Staubli VAL3: LEFTPOS.pgx

public program leftPos(string x_sItem, num x_nLength, string& x_sResult[])
  local num i
  local num l_nLength
  local string l_sItem
begin
  //-----------------------------------------------------------------------
  //Header begin
  //Description of program
  //  This program allows to keep x_nLength characters of a string from
  //  the left side.
  //  The characters after x_nLength on the right side will be truncated.
  //
  //Input parameters
  //  string x_sItem :
  //    role : string that you wan to cut
  //  num x_nLength :
  //    role : Length of the characters that you want to keep
  //
  //Output parameters
  //  string x_sResult :
  //    role : string truncated
  //
  //Example
  //  call leftPos("Staubli Robotics",7,sResult)
  //  put(sResult) //Displays "Staubli"
  //
  //History
  //  Creation : 28-04-08 - f.Rob
  //Header end
  //-----------------------------------------------------------------------
  l_sItem=x_sItem
  //Divide the string...
  if len(l_sItem)!=getDisplayLen(l_sItem) and x_nLength!=0
    for i=0 to len(x_sItem)-1
      l_nLength=l_nLength+getDisplayLen(left(l_sItem,1))
      l_sItem=right(l_sItem,len(l_sItem)-1)
      if l_nLength==x_nLength
        x_sResult=left(x_sItem,i+1)
        return
      else
        if l_nLength>x_nLength
          x_sResult=left(x_sItem,i)
          return
        endIf
      endIf
    endFor
  endIf
  x_sResult=left(x_sItem,x_nLength)
end
